FUNCTION_BLOCK CU030GroundTask EXTENDS CUBaseGround IMPLEMENTS ICUTask

Run();

METHOD DataEntityDiscard
VAR_INPUT	
	inStepID : INT;
	EntityId : STRING(255);
END_VAR
IF (Step(inStepID, TRUE, 'DISCARD ENTITY')) THEN	
    //-------------------------------------		
	IF(Station.ProcessDataManager.Exists(EntityId).Done) THEN
		IF(Station.ProcessDataManager._idExistsTask.Exists) THEN
			StepCompleteWhen(THIS^.Station.EntityFlowDiscard(EntityId, Station.ProcessDataManager.Data.CU030.Header).Done);
		ELSE
			CompleteStep();
		END_IF
	END_IF;					   		    				
    //-------------------------------------
END_IF
END_METHOD

(*~
	<docu>
		<summary>
			Main method of the sequener. Custom code needs to be placed here. The sequencer is executed by call of **Instance.Run()** method.
			This method is abstract, and it must be overridden in derived block.
		</summary>
	</docu>
~*)
METHOD PROTECTED Main : BOOL
IF (Step(100, TRUE, 'STOPPING OTHER MODES')) THEN
	Station.AutomatTask.ResetCycleTime();//here we can reset averages values of CT
	Station.AutomatTask.Restore();
	Station.ManualTask.Restore();
	Station.ProcessDataManager.Restore();
	Station.AutomatTask.HideAllDialogs();
	Station.GroupInspection.Restore();// hide all dialogs 
    StepCompleteWhen(TRUE);
END_IF

IF (Step(200, TRUE, 'STOPPING OTHER MODES')) THEN	
//	---------------------------------------------------
	
	Station.AutomatTask.ResetCycleTime();
	Station.ProductionPlanerTask.Restore();
	Station.Components.PairTagTask.Restore();
	
	Messenger.Info('INFO MESSAGE');
	
    StepCompleteWhen(THIS^._currentStep.Duration > T#500MS);
//	---------------------------------------------------
END_IF

DataEntityDiscard(5000, THIS^.Station.ProcessDataManager.Data._EntityId);

IF (Step(10000, TRUE, 'LAST STEP')) THEN	
	//---------------------------------------------------
	_groundDone := TRUE;
	THIS^._task.DoneWhen(_groundDone);
	//---------------------------------------------------
END_IF
END_METHOD

METHOD PUBLIC OnStart
SUPER^.OnStart();
Station.AutomatTask.Restore();
Station.ManualTask.Restore();
Station.GroundTask.CancelGround();
END_METHOD

PROPERTY Station : REFERENCE TO CU030
GET
VAR
    _station : POINTER TO CU030;
END_VAR
IF __QUERYPOINTER(Parent, _station) THEN // Check if _Parent is Station001
    Station REF= _station^;              // If the check is successful dereference a pointer. simlar to THIS^ or SUPER^
END_IF
END_GET
END_PROPERTY

END_FUNCTION_BLOCK

(* stored: Version 1.1.0.1
   POU CU030GroundTask: Id {98e262ef-df52-4ce0-bfe2-6a26f1bf9478}, SpecialFunc None
   Folder DataOperations: Id {6de64a46-4f50-43c1-ae7c-4d4f99c79759}
   Method DataEntityDiscard: Id {67c4e98b-90b8-4533-9048-95ebd71615ab}
   Method Main: Id {6de1a2fe-d2fe-4de4-ae32-3e9a075fdd60}
   Method OnStart: Id {96e5ed22-8b55-4651-b085-7aecd3e4a3b8}
   Property Station: Id {7a0c32f3-63fd-4f54-8817-d2a2aa6c6e8b}
   Get Get: Id {e6d03756-ac12-4bd0-b29c-ddda1051b057} *)
